{attribute 'qualified_only'}
VAR_GLOBAL
//motor global 
	motor1: motorDUT; 
	motor2: motorDUT;
// GUI
	StartStop: BOOL; //start and stop process  
	systemOK: bool; //true if system is ready
END_VAR

(* stored: Version 1.1.0.1, ProductVersion 3.1.4024.12
   GVL GVL: Id {eb1c2fde-2fa8-418a-8f7f-81f033c5433b} *)
